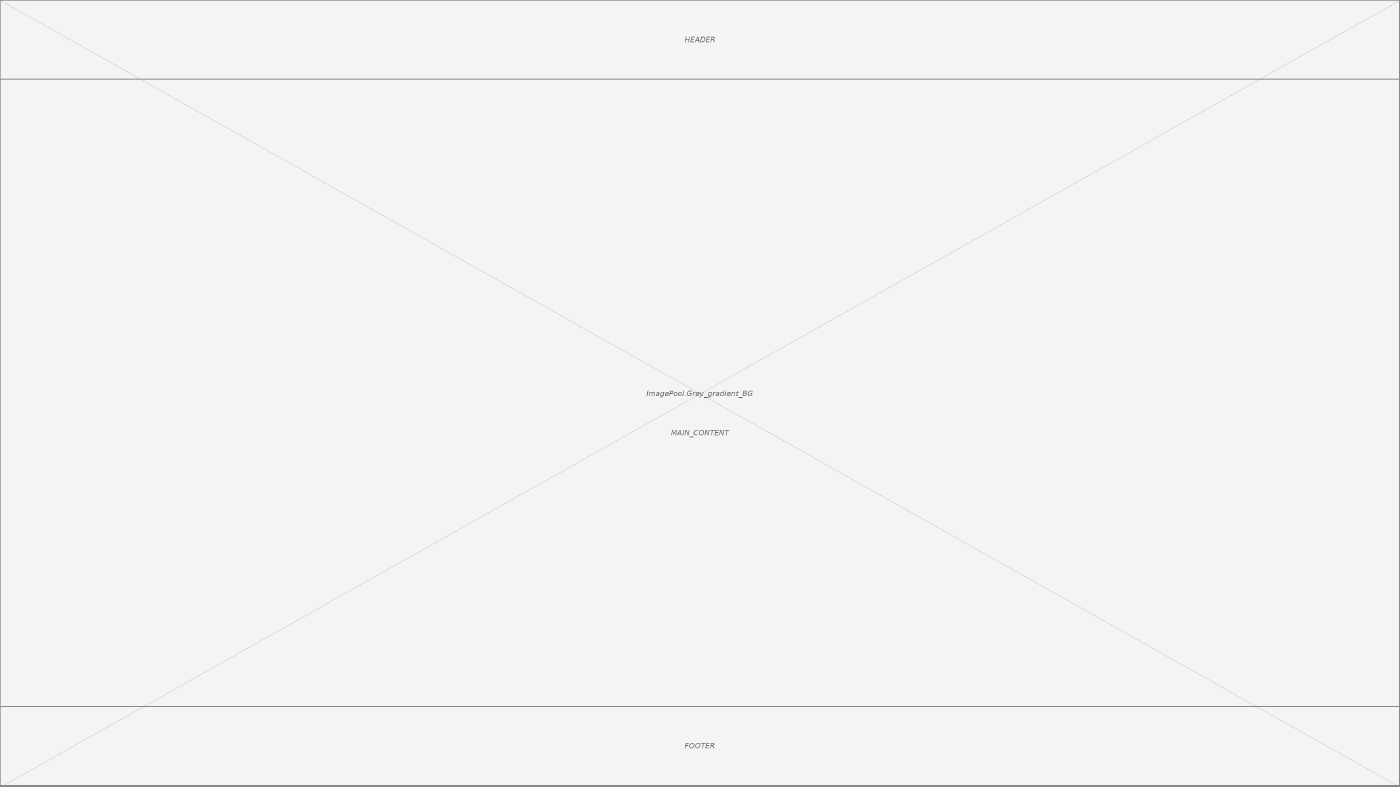
VISUALIZATION MAIN_PAGE  // 1920x1080
    Rectangle (0,0 1920x1080)
    Image (0,0 1920x1080), image: ImagePool.Grey_gradient_BG
    Frame (0,108 1920x972)
        shows MAIN_CONTENT()
        shows KUKA_PROG()
        shows HEADER()
    Frame (0,0 1920x109)
        shows HEADER()
        shows KUKA_PAGE()
        shows KUKA_PROG_CONTENT()
        shows MAIN_CONTENT()
        shows KUKA_IO_CONTENT()
    Frame (0,969 1920x109)
        shows FOOTER()
END_VISUALIZATION

(* stored: Version 1.1.0.1, ProductVersion 3.1.4024.12
   Visu MAIN_PAGE: Id {88eaab8b-c2f1-465f-93c8-1f4b9b2850db} *)
